// TIA Portal V21 export
TYPE "Std_RicettaUniverale"
   STRUCT
      Lavoro : "Std_RicettaUniverale_Prm";
      Modifica : "Std_RicettaUniverale_Prm";
      Originali { S7_SetPoint := 'True'} : "Std_RicettaUniverale_Prm";
      Archivio : Array[0.."K_NumRicettaPerMacchina"] of "Std_RicettaUniverale_Prm";
      Hmi : Struct
         NumDatoRicettaBool : Int;
         NumDatoRicettaReal : Int;
         CodiceMacchinario : Int;
         Indice_Selezionata : Int;
         Indice_RicettaAttuale : Int;
         Indice_CopiaDa : Int;
         Indice_CopiaIn : Int;
         Esegui_Annulla : Bool;
         Esegui_Carica : Bool;
         Esegui_Salva : Bool;
         Esegui_Copia : Bool;
         Esegui_ModificaRicettaInLavoro : Bool;
         Esegui_ModificaRicettaInArchivio : Bool;
         InCorso_ModificaRicettaInLavoro : Bool;
         InCorso_ModificaRicettaInArchivio : Bool;
         Scelta_CopiaDa : Bool;
         Scelta_CopiaIn : Bool;
         RichiediSalvataggio : Bool;
         FocusArchivio : Bool;
         AvviaCopia : Bool;
         AbilitaCarica : Bool;
         AbilitaCopia : Bool;
         Abilita_ModificaRicettaInLavoro : Bool;
         Abilita_ModificaRicettaInArchivio : Bool;
         MemoOldSelezione : Int;
         MostraOriginali : Bool;
         Archivio : Struct
            AbilitaIncrementoRicetta : Bool;
            AbilitaDecrementoRicetta : Bool;
            IndiceFormatoVisualizzato : Int;
            IndiceHmi : Array[0.."K_RicetteAdHmi"] of Int;
            NomeHmi : Array[0.."K_RicetteAdHmi"] of String;
            SelezioneHmi : Array[0.."K_RicetteAdHmi"] of Bool;
         END_STRUCT;
      END_STRUCT;
      Out : Struct
         ScriviDatiLagica : Bool;
      END_STRUCT;
      Allarmi : Struct
         "A" { S7_SetPoint := 'True'} : Array[0.."K_NumAllarmiPerRicette"] of "Std_PrmAllarmeStd";
         WordHMI : Word := 16#0000;
      END_STRUCT;
   END_STRUCT;
   // Allarmi."A"[0..2].Stato := FALSE;
   // Allarmi."A"[0..2].EnWarnHmi := FALSE;
   // Allarmi."A"[0..2].EnCadutaCiclo := FALSE;
END_TYPE
